// TIA Portal V16 export
// export: Created 2023-03-03T12:40:02.4425328Z, ExportSetting WithDefaults, DisplayName Totally Integrated Automation Portal, DisplayVersion V16 Update 3, DisplayName TIA Portal Version Control Interface, DisplayVersion V16 Update 2, DisplayName TIA Portal Openness, DisplayVersion V16 Update 3, DisplayName STEP 7 Professional, DisplayVersion V16 Update 3, DisplayName STEP 7 Safety, DisplayVersion V16, DisplayName WinCC Professional, DisplayVersion V16 Update 3
VAR_GLOBAL   // PLC tag table "FC19511_Test"
   SIM001_TRIGGER AT %M900.0 : Bool;   // Simulation Trigger Signal
   SIM001_OUTPUT AT %MD910 : Real;   // Simulation Output
   SIM001_INPUT AT %MD902 : Real;   // Simulation Input
   SIM001_Type AT %MW906 : Int;   // 0 = Step, 1 = Ramp, 2 = Sinusoid
   "Counter" AT %MW908 : Int;   // 100ms Counter
END_VAR
